FUNCTION_BLOCK Test_ErrorIdToString EXTENDS T_UnitTestBase
VAR_INPUT
END_VAR
VAR_OUTPUT
END_VAR
VAR
	Assertion : T_Assertion;
END_VAR

{attribute 'analysis' := '-33'} // inhibit unused variable warning
METHOD RunTest
VAR_OUTPUT
    TestCompleted : BOOL;
    TestFailed    : BOOL;
END_VAR
TestFailed S= NOT Assertion.AssertEquals_STRING(Source    := TestName,
                             Expected     := 'Error 0x12BD',
                              Actual       := F_ErrorIdToString(16#12BD),
                              VariableName := 'F_ErrorIdToString(16#12BD)');

TestFailed S= NOT Assertion.AssertEquals_STRING(Source    := TestName,
                             Expected     := 'Error 0x12345678',
                              Actual       := F_ErrorIdToString(16#12345678),
                              VariableName := 'F_ErrorIdToString(16#12345678)');

TestFailed S= NOT Assertion.AssertEquals_STRING(Source    := TestName,
                             Expected     := 'Error 0x00FF',
                              Actual       := F_ErrorIdToString(16#FF),
                              VariableName := 'F_ErrorIdToString(16#FF)');

TestFailed S= NOT Assertion.AssertEquals_STRING(Source    := TestName,
                             Expected     := 'Error 0x0011 - No debugging available',
                              Actual       := F_ErrorIdToString(16#11),
                              VariableName := 'F_ErrorIdToString(16#11)');

TestCompleted := TRUE;
END_METHOD

END_FUNCTION_BLOCK

(* stored: Version 1.1.0.1, ProductVersion 3.1.4024.12
   POU Test_ErrorIdToString: Id {932a14fe-2c3a-4e26-b5ff-ff299c485b65}, SpecialFunc None
   Method RunTest: Id {323e7f4e-87f5-4973-b46e-7a12c295ef73} *)
